FUNCTION_BLOCK E_D_FF (* Data latch (d) flip flop *)
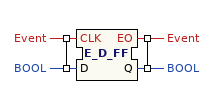
  EVENT_INPUT
    CLK WITH D; (* Clock *)
  END_EVENT
  EVENT_OUTPUT
    EO WITH Q; (* Triggered if clock results in a change of Q *)
  END_EVENT
  VAR_INPUT
    D : BOOL; (* Value to latch *)
  END_VAR
  VAR_OUTPUT
    Q : BOOL; (* Latched value *)
  END_VAR
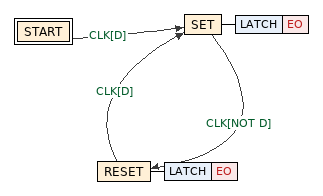
  EC_STATES
    START; (* Initial State *)
    SET : LATCH -> EO; (* Initialization *)
    RESET : LATCH -> EO;
  END_STATES
  EC_TRANSITIONS
    START TO SET := CLK[D];
    SET TO RESET := CLK[NOT D];
    RESET TO SET := CLK[D];
  END_TRANSITIONS
  ALGORITHM LATCH IN ST: (* new algorithm *)
Q := D;
  END_ALGORITHM
END_FUNCTION_BLOCK
